# EPICS alarm handler configuration: mps_database/bareTest/alarms/areas/mpln_ltuh_mp03.alhConfig
GROUP NULL MPLN:LTUH:MP03:1
$ALIAS MPS Link Node 132
$GUIDANCE
LTUH MPS
   Group Name: MPLN:LTUH:MP03:1
   Summary PV:  MPLN:LTUH:MP03:1:STATSUMY
$END
CHANNEL  MPLN:LTUH:MP03:1    MPLN:LTUH:MP03:1:MPS_EN_RBV		-----
CHANNEL  MPLN:LTUH:MP03:1    MPLN:LTUH:MP03:1:LC1_MODE_RBV		-----
